// TIA Portal V17 export
// export: Created 2022-07-20T07:02:16.76792Z, ExportSetting WithDefaults, DisplayName Totally Integrated Automation Portal, DisplayVersion V17, DisplayName TIA Portal Openness, DisplayVersion V17, DisplayName TIA Portal Version Control Interface, DisplayVersion V17, DisplayName SINAMICS Startdrive Advanced, DisplayVersion V17, DisplayName SINAMICS Startdrive G130, G150, S120, S150, SINAMICS MV, S210, DisplayVersion V17, DisplayName SINAMICS Startdrive G110M, G120, G120C, G120D, G120P, G115D, DisplayVersion V17, DisplayName STEP 7 Professional, DisplayVersion V17, DisplayName STEP 7 Safety, DisplayVersion V17, DisplayName WinCC Advanced, DisplayVersion V17
FUNCTION_BLOCK "FB10032_CalcCam"   // FB10032, LAD
{ S7_Optimized_Access := 'TRUE' }
VERSION : 0.1
// stored: AutoNumber false, IsIECCheckEnabled false, IsRetainMemResEnabled false, MemoryReserve 100, SetENOAutomatically false, UDAEnableTagReadback false
   VAR_INPUT
      Execute : Bool;
      Reset : Bool;
      NbPoint : Int;
   END_VAR
   VAR_OUTPUT
      Done { ExternalAccessible := 'False'; ExternalVisible := 'False'; ExternalWritable := 'False'} : Bool;   // TRUE: Commanded action has been completed successfully
      Busy { ExternalAccessible := 'False'; ExternalVisible := 'False'; ExternalWritable := 'False'} : Bool;   // TRUE: FB is not finished and new output values can be expected
      Error { ExternalAccessible := 'False'; ExternalVisible := 'False'; ExternalWritable := 'False'} : Bool;   // Rising edge informs that an error occurred during the execution of
      ErrorID : Word;
      Status : Word;
   END_VAR
   VAR_IN_OUT
      Profile : Array[*] of "LCamHdl_typeBasicPoint";
      Cam : TO_Cam;
   END_VAR
   VAR
      statExecuteOld { ExternalAccessible := 'False'; ExternalVisible := 'False'; ExternalWritable := 'False'} : Bool;   // Old value of execute for edge detection
      statExecute : Bool;
      statDone { ExternalAccessible := 'False'; ExternalVisible := 'False'; ExternalWritable := 'False'} : Bool;   // Static value for output done
      statBusy { ExternalAccessible := 'False'; ExternalVisible := 'False'; ExternalWritable := 'False'} : Bool;   // Static value for output busy
      statNbOfElements { S7_SetPoint := 'True'} : Int;
      statDiagnostics { ExternalWritable := 'False'} : "LCamHdl_typeDiagnostics";   // Diagnostics information of FB
      statStatus { S7_SetPoint := 'True'} : Word;
      statErrorID : Word;
      statError : Bool;
      LCamHdl_CreateCamBasic_Instance { S7_SetPoint := 'True'} : "LCamHdl_CreateCamBasic";
   END_VAR
   VAR CONSTANT
      STATUS_NO_CALL : Word := 16#7000;   // No call of FB
      STATUS_CHECK_CONFIGURATION : Word := 16#7001;
      STATUS_CONFIGURATION_CHECKED : Word := 16#7002;
      STATUS_EXECUTION_CALCUL : Word := 16#7003;
      STATUS_EXECUTION_FINISHED : Word := 16#7004;   // Execution finished without errors
      STATUS_ERROR : Word := 16#7999;
      ERR_NOERRROR : Word := 16#0000;
      ERR_CONFIGURATION : Word := 16#9000;
      ERR_CALCUL : Word := 16#9001;
      ERR_ABORT : Word := 16#9002;
   END_VAR
BEGIN

REGION Network 1 (SCL): (** COMMENTS **)
   //==========================================================================================
   // SIEMENS SAS      RC-FR DI FA APC
   // ------------------------------------------------------------------------------------------
   // Library:         LAPCFR
   // Tested with:     S7-1515TF
   // FW Version:      2.8
   // Engineering:     TIA Portal V16
   // Restrictions:    ---
   // Requirements:    Motion Control Library V5.0
   //------------------------------------------------------------------------------------------
   // Description:     Cam calculation via profile in advanced elements
   //------------------------------------------------------------------------------------------
   // Change log table:
   // Version    Date          Expert in charge    Changes applied
   // 01.00.00   2020.05.25    RTO                 First released version
   //===========================================================================================
END_REGION

REGION Network 2 (SCL): (** SEQUENCE**)
   //** Initialization **//
   IF #Execute AND NOT #statExecuteOld AND NOT #statBusy
   THEN

       #statExecute := FALSE;
       #statStatus := #STATUS_CHECK_CONFIGURATION;
       #statBusy := TRUE;
       #statError := FALSE;
       #statErrorID := #ERR_NOERRROR;

       IF #NbPoint < 1
       THEN
           #statErrorID := #ERR_CONFIGURATION;
           #statError := TRUE;
       ELSE
           #statStatus := #STATUS_CONFIGURATION_CHECKED;
       END_IF;

       #statNbOfElements := #NbPoint;

   END_IF;

   //** Executed **//
   IF #Execute AND #statStatus = #STATUS_CONFIGURATION_CHECKED THEN
       #statExecute := TRUE;
       #statStatus := #STATUS_EXECUTION_CALCUL;
   END_IF;

   //** Aborted  **//
   IF NOT #Execute AND #statExecuteOld AND #statStatus <> #STATUS_EXECUTION_FINISHED THEN
       #statErrorID := #ERR_ABORT;
       #statError := TRUE;
       #statExecute := FALSE;
       #statBusy := FALSE;
   END_IF;

   //** Done **//
   IF NOT #Execute AND #statExecuteOld AND #statStatus = #STATUS_EXECUTION_FINISHED THEN
       #statStatus := #STATUS_NO_CALL;
   END_IF;
END_REGION

REGION Network 3 (SCL): (** ERROR **)
   //** Abort **//
   IF #statError THEN
       //#statExecute := FALSE;
       #statBusy := FALSE;
   END_IF;

   //** Reset **//
   IF #Reset THEN
       #statErrorID := #ERR_NOERRROR;
       #statError := FALSE;
   END_IF;
END_REGION

REGION Network 4: (** CALL CALCUL BLOCK **)
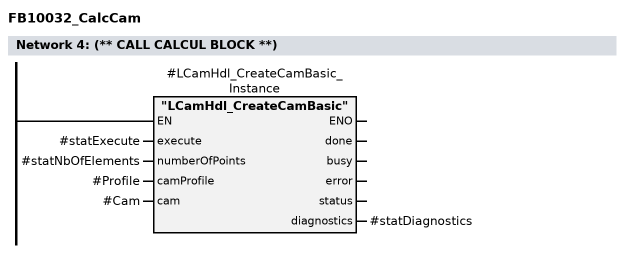
   RUNG wire#powerrail
      #LCamHdl_CreateCamBasic_Instance(execute := #statExecute, numberOfPoints := #statNbOfElements, camProfile := #Profile, cam := #Cam, done =>, busy =>, error =>, status =>, diagnostics => #statDiagnostics)
   END_RUNG
   // the same network as SCL:
   #LCamHdl_CreateCamBasic_Instance(execute := #statExecute,   // "LCamHdl_CreateCamBasic"
                           numberOfPoints := #statNbOfElements,
                           camProfile := #Profile,
                           cam := #Cam,
                           diagnostics => #statDiagnostics);
END_REGION

REGION Network 5 (SCL): (** CALCUL BLOCK STATUS**)
   IF #LCamHdl_CreateCamBasic_Instance.error THEN
       #statErrorID := #ERR_CALCUL;
       #statError := TRUE;
   END_IF;

   IF #LCamHdl_CreateCamBasic_Instance.done THEN
       #statStatus := #STATUS_EXECUTION_FINISHED;
       #statExecute := FALSE;
       #statBusy := FALSE;
   END_IF;
END_REGION

REGION Network 6 (SCL): (** OUTPUT **)
   #Error := #statError;
   #ErrorID := #statErrorID;
   #Done := #statStatus = #STATUS_EXECUTION_FINISHED;
   #Busy := #statBusy;
   #statExecuteOld := #Execute;
   #Status := #statStatus;
END_REGION
END_FUNCTION_BLOCK
